FUNCTION_BLOCK SpeedTrigger EXTENDS Objective
VAR

	{attribute 'hide'}
	internalThresholdVelocity	: LREAL;	

END_VAR

{attribute 'monitoring' := 'variable'}
PROPERTY CurrentMover : REFERENCE TO Mover
GET
VAR
	i	: USINT;
END_VAR

CurrentMover 	REF= 0;

FOR i := 0 TO SIZEOF( TrackedMovers[0] ) / SIZEOF( TrackedMovers ) - 1 DO
	
	IF TrackedMovers[i] <> 0 AND_THEN ( ABS(TrackedMovers[i]^.AxisReference.NcToPlc.ActVelo) >= ThresholdVelocity ) THEN
		CurrentMover	REF= TrackedMovers[i]^;
	END_IF
		
END_FOR
END_GET
END_PROPERTY

{attribute 'monitoring' := 'variable'}
PROPERTY MoverInVelocity : BOOL
GET
VAR
	i	: USINT;
END_VAR

MoverInVelocity		:= FALSE;

FOR i := 0 TO GVL.NUM_MOVERS - 1 DO
	
	IF TrackedMovers[i] <> 0 AND_THEN ( ABS(TrackedMovers[i]^.AxisReference.NcToPlc.ActVelo) >= ThresholdVelocity ) THEN
		MoverInVelocity		:= TRUE;		
	END_IF
	
END_FOR
END_GET
END_PROPERTY

PROPERTY ThresholdVelocity : LREAL
GET


	ThresholdVelocity		:= internalThresholdVelocity;
END_GET
SET



	internalThresholdVelocity		:= ThresholdVelocity;
END_SET
END_PROPERTY

END_FUNCTION_BLOCK

(* stored: Version 1.1.0.1, ProductVersion 3.1.4024.9
   POU SpeedTrigger: Id {ceb84e98-9bb3-44af-9526-f95d6c0344e5}, SpecialFunc None
   Folder Methods: Id {509b1e5d-b79a-449e-ba49-e162eb42b6fc}
   Folder Properties: Id {dbd68162-6541-404e-b05a-0fec2a8ff4c5}
   Property CurrentMover: Id {7f0937a7-bed5-48ff-acf8-6553ecfccecb}
   Get Get: Id {579026c0-dbc9-45df-a0d9-58debaf1382a}
   Property MoverInVelocity: Id {7c83a599-b5f9-45c9-9131-e8a02b23529a}
   Get Get: Id {2ea072c0-2f9e-44bb-b822-47a0341f43bf}
   Property ThresholdVelocity: Id {1f1a632c-f4e8-446f-9260-5f7e4c9c9017}
   Get Get: Id {02cc51fd-1552-49da-a92a-6edba1c95096}
   Set Set: Id {dfd5cdd4-fa57-4379-b145-1e679363cb0e} *)
